(****************************************************************************)
(*							Beckhoff Automation Poland						*)
(*							F_4BYTES_TO_DWORD v1							*)
(*									21.11.2013								*)
(*					Funkcja zamieniająca 4 zmienne typu BYTE na DWORD 		*)
(*__________________________________________________________________________*)
FUNCTION F_4BYTES_TO_DWORD : DWORD
VAR_INPUT
	BByte0		: BYTE;
	BByte1		: BYTE;
	BByte2		: BYTE;
	BByte3		: BYTE;
END_VAR

F_4BYTES_TO_DWORD := BByte3 *16#1000000 + BByte2 *16#10000 + BByte1 *16#100 + BByte0;

END_FUNCTION

(* stored: Version 1.1.0.1, ProductVersion 3.1.4026.13, FileIdentifier 3c693ebecac7968ca8616392d02ea38248d1937a, FileSignature 2415682906437b1923cad7677591ba8500f953069697d6e782715db7a26392d26519c69a69fd94f0d068ff3c315e0374c7d314b8af84f5f2ad5c01445ddf13e9c0b2303b1b9f7ed6871f4c8ff24bc47af64c9df43e3223a785d1f53829078c391d03e8df7a2ba9543ef2dccb3fde91e848bd489bdde3bf7b28f8a6bb4ed61ca0d10cb8275c6eef8fe592ddc064089fec436a5a8fe3dfbeee484a420ff6c36734dd68f5a97d1869d5b7aa41f46c62a0774a68f476a2413f07984d96f4ec13accb274d66badc731a8bdad3fcdb832db20f04f348ffd30061f2d5f6c30f65e07eb9ec1ba9e5e96eb67016e7d81b428f40a3877a013d128e4b35d2cd763011fa50af
   POU F_4BYTES_TO_DWORD: Id {cac8c25e-a34f-4816-9472-a6a481f47fb3}, SpecialFunc None *)
